VAR_GLOBAL
	SolderingStart:BOOL;
END_VAR

(* stored: Version 1.1.0.1, ProductVersion 3.1.0.36
   GVL GVL_Soldering: Id {c344cd74-9d73-4cdc-8729-dddef89ca58f} *)
